# EPICS substitutions: apps/monitorApp/Db/bonner-spheres.substitutions
file "db/bonner-sphere.db" {
    pattern { P }
    { B_BS1_ }
    { B_BS2_ }
    { B_BS3_ }
    { B_BS4_ }
    { B_BS5_ }
    { B_BS6_ }
}
